// TIA Portal project "Level Control - Pump Start and Stop Ladder Logic" (V17)
// Level Control - Pump Start and Stop Ladder Logic
// If the low level sensor detects that the tank is low, then the pump will run for 20 seconds.
// If the high level sensor detects that the tank is full, the pump should stop for 30 seconds.

(* hardware
DEVICE "S7-1200 station_1"  S7-1200 Station
   slot 0: "Rack_0"  S7-1200 Rack  Rack  V1.0
   slot 1: "PLC_1"  CPU 1212C DC/DC/DC  6ES7 212-1AE40-0XB0  V4.5
*)

// ===== PLC "PLC_1"  CPU 1212C DC/DC/DC =====

VAR_GLOBAL   // PLC tag table "Default tag table"
   "PB" AT %I0.0 : Bool;
   "Low level sensor" AT %I0.1 : Bool;
   "High level sensor" AT %I0.2 : Bool;
   "Pump motor" AT %Q0.0 : Bool;
   "Tag_1" AT %M0.0 : Bool;
END_VAR

// folder: System blocks/Program resources

DATA_BLOCK "IEC_Timer_0_DB"   // DB1
{ S7_Optimized_Access := 'TRUE' }
AUTHOR : Simatic
FAMILY : IEC
NAME : IEC_TMR
VERSION : 1.0
// stored: InstanceOfName IEC_TIMER
"IEC_TIMER"
BEGIN
END_DATA_BLOCK

DATA_BLOCK "IEC_Timer_0_DB_1"   // DB2
{ S7_Optimized_Access := 'TRUE' }
AUTHOR : Simatic
FAMILY : IEC
NAME : IEC_TMR
VERSION : 1.0
// stored: InstanceOfName IEC_TIMER
"IEC_TIMER"
BEGIN
END_DATA_BLOCK

// folder: (top level)

ORGANIZATION_BLOCK "Main"   // OB1, LAD, ProgramCycle
TITLE = "Main Program Sweep (Cycle)"
{ S7_Optimized_Access := 'TRUE' }
VERSION : 0.1
   VAR_INPUT
      Initial_Call : Bool;   // Initial call of this OB
      Remanence : Bool;   // =True, if remanent data are available
   END_VAR
BEGIN

REGION Network 1
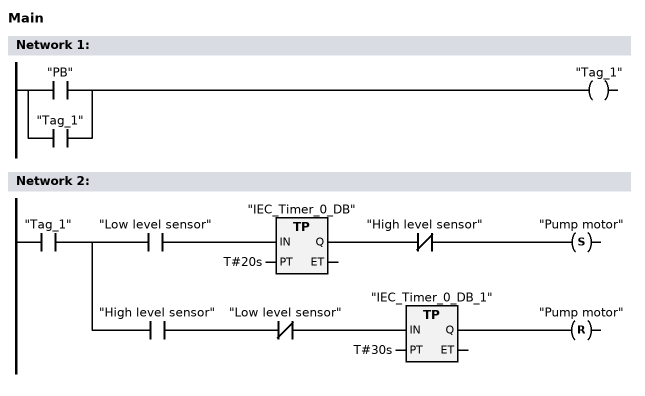
   RUNG wire#powerrail
      Contact( "PB" )
      wire#w1
      Coil( "Tag_1" )
   END_RUNG
   RUNG wire#powerrail
      Contact( "Tag_1" )
   END_RUNG wire#w1
   // the same network as SCL:
   "Tag_1" := "PB" OR "Tag_1";
END_REGION

REGION Network 2
   "IEC_Timer_0_DB".TP(IN := "Tag_1" AND "Low level sensor", PT := T#20s);
   IF "IEC_Timer_0_DB".Q AND NOT "High level sensor" THEN "Pump motor" := TRUE; END_IF;
   "IEC_Timer_0_DB_1".TP(IN := "Tag_1" AND "High level sensor" AND NOT "Low level sensor", PT := T#30s);
   IF "IEC_Timer_0_DB_1".Q THEN "Pump motor" := FALSE; END_IF;
END_REGION
END_ORGANIZATION_BLOCK